FUNCTION_BLOCK FB_TP (* standard timer function block (pulse) *)
  (* Standard: 61131-3; Classification: standard timer function block; Description: Copyright (c) 2011 TU Wien ACIN This program and the accompanying materials are made available under the terms of the Eclipse Public License 2.0 which is available at https://www.eclipse.org/legal/epl-2.0/ SPDX-License-Identifier: EPL-2.0 *)
  (* Version 3.0, 2025-04-14, Patrick Aigner, changed package *)
  (* Version 1.0, 2011-06-21, Monika Wenger, TU Wien ACIN *)
  PACKAGE iec61131::timers;
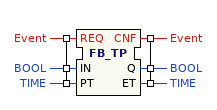
  EVENT_INPUT
    REQ WITH IN, PT; (* Service Request *)
  END_EVENT
  EVENT_OUTPUT
    CNF WITH Q, ET; (* Confirmation of Requested Service *)
  END_EVENT
  VAR_INPUT
    IN : BOOL; (* Input *)
    PT : TIME; (* Pulse time *)
  END_VAR
  VAR_OUTPUT
    Q : BOOL; (* output *)
    ET : TIME; (* elapse time *)
  END_VAR
END_FUNCTION_BLOCK
